{attribute 'GeneratedUsingTerminal: EK1122-0000-0018'}
{attribute addProperty BoxType "EK1122-0000-0018"}
{attribute addProperty Id "Beckhoff_EP7xxxsub_EK1100EK1100_1FC0878B2A_0001_EP7041_0002_0016EP7041_7A2D1F1A44A_0002_EP7041_0002_0017EP7041_7A2D1F1A44A_0003_EP7041_0002_0018EP7041_5C004D4E45A_0004_EP7041_0002_0019EP7041_5C004D4E45A_0005_EP7041_0002_0020EP7041_5C004D4E45A_0006_EP7041_0002_0021EP7041_5C004D4E45A_0007_EP7041_0002_0022EP7041_5C004D4E45A_0008_EP7041_0002_0023EP7041_5C004D4E45A_0009_EP7041_0002_0024EP7041_5C004D4E45A_0010_EP7041_0002_0025EP7041_5C004D4E45A_0011_EP7041_1002_0017EP7041_7A2D1F1A44A_0012_EP7041_1002_0018EP7041_5C004D4E45A_0013_EP7041_1002_0019EP7041_5C004D4E45A_0014_EP7041_1002_0020EP7041_5C004D4E45A_0015_EP7041_1002_0021EP7041_5C004D4E45A_0016_EP7041_1002_0022EP7041_5C004D4E45A_0017_EP7041_1002_0023EP7041_5C004D4E45A_0018_EP7041_1002_0024EP7041_5C004D4E45A_0019_EP7041_1002_0025EP7041_5C004D4E45A_0020_EP7041_2002_0016EP7041_5C004D4E45A_0021_EP7041_2002_0019EP7041_5C004D4E45A_0022_EP7041_2002_0020EP7041_5C004D4E45A_0023_EP7041_2002_0021EP7041_5C004D4E45A_0024_EP7041_2002_0022EP7041_5C004D4E45A_0025_EP7041_2002_0023EP7041_5C004D4E45A_0026_EP7041_2002_0024EP7041_5C004D4E45A_0027_EP7041_2002_0025EP7041_5C004D4E45A_0028_EP7041_3002_0016EP7041_B6E6359B46A_0029_EP7041_3002_0017EP7041_B6E6359B46A_0030_EP7041_3002_0018EP7041_B6E6359B46A_0031_EP7041_3002_0019EP7041_B6E6359B46A_0032_EP7041_3002_0020EP7041_B6E6359B46A_0033_EP7041_3002_0021EP7041_B6E6359B46A_0034_EP7041_3002_0022EP7041_B6E6359B46A_0035_EP7041_3102_0016EP7041_B6E6359B46A_0036_EP7041_3102_0017EP7041_B6E6359B46A_0037_EP7041_3102_0022EP7041_B6E6359B46A_0038_EP7047_1032_0021EP7047_B6E6359B46A_0039_EP7211_0034_0029EP7211_91DE43F025A_0040_EP7211_0034_0030EP7211_0985306B26A_0041_EP7211_0034_0031EP7211_0985306B26A_0042_EP7211_0034_0032EP7211_0985306B26A_0043_EP7211_0035_0029EP7211_24495B2825A_0044_EP7211_0035_0030EP7211_24495B2825A_0045_EP7211_0035_0031EP7211_24495B2825A_0046_EP7211_0035_0032EP7211_24495B2825A_0047_EP7342_0002_0016EP7342_A970B60778A_0048_EP7342_0002_0017EP7342_A970B60778A_0049_EP7342_0002_0018EP7342_A970B60778A_0050_EP7342_0002_0019EP7342_A970B60778A_0051_EP7342_0002_0020EP7342_A970B60778A_0052_EP7342_0002_0021EP7342_A970B60778A_0053_EP7342_0002_0022EP7342_A970B60778A_0054_EP7402_0057_0017A_0054_EP7402_0057_0017_470DA1C691"}
{attribute addProperty CRC "1867209835"}
{attribute addProperty Size "2560"}
TYPE Beckhoff_EP7xxxEK1122_6F4B5C6B EXTENDS EK1122_1FC0878B :
STRUCT
	{attribute addProperty Name "Beckhoff_EP7xxxsub_EK1100"}
	{attribute addProperty PreviousPort "Beckhoff EP7xxxEK1122 : D"}
	Beckhoff_EP7xxxsub_EK1100 : EK1100_1FC0878B;
	{attribute addProperty Name "A_0001_EP7041_0002_0016"}
	{attribute addProperty PreviousPort "Beckhoff EP7xxxsub EK1100 : C"}
	A_0001_EP7041_0002_0016 : EP7041_7A2D1F1A;
	{attribute addProperty Name "A_0002_EP7041_0002_0017"}
	{attribute addProperty PreviousPort "A_0001(EP7041-0002-0016) : B"}
	A_0002_EP7041_0002_0017 : EP7041_7A2D1F1A;
	{attribute addProperty Name "A_0003_EP7041_0002_0018"}
	{attribute addProperty PreviousPort "A_0002(EP7041-0002-0017) : B"}
	A_0003_EP7041_0002_0018 : EP7041_5C004D4E;
	{attribute addProperty Name "A_0004_EP7041_0002_0019"}
	{attribute addProperty PreviousPort "A_0003(EP7041-0002-0018) : B"}
	A_0004_EP7041_0002_0019 : EP7041_5C004D4E;
	{attribute addProperty Name "A_0005_EP7041_0002_0020"}
	{attribute addProperty PreviousPort "A_0004(EP7041-0002-0019) : B"}
	A_0005_EP7041_0002_0020 : EP7041_5C004D4E;
	{attribute addProperty Name "A_0006_EP7041_0002_0021"}
	{attribute addProperty PreviousPort "A_0005(EP7041-0002-0020) : B"}
	A_0006_EP7041_0002_0021 : EP7041_5C004D4E;
	{attribute addProperty Name "A_0007_EP7041_0002_0022"}
	{attribute addProperty PreviousPort "A_0006(EP7041-0002-0021) : B"}
	A_0007_EP7041_0002_0022 : EP7041_5C004D4E;
	{attribute addProperty Name "A_0008_EP7041_0002_0023"}
	{attribute addProperty PreviousPort "A_0007(EP7041-0002-0022) : B"}
	A_0008_EP7041_0002_0023 : EP7041_5C004D4E;
	{attribute addProperty Name "A_0009_EP7041_0002_0024"}
	{attribute addProperty PreviousPort "A_0008(EP7041-0002-0023) : B"}
	A_0009_EP7041_0002_0024 : EP7041_5C004D4E;
	{attribute addProperty Name "A_0010_EP7041_0002_0025"}
	{attribute addProperty PreviousPort "A_0009(EP7041-0002-0024) : B"}
	A_0010_EP7041_0002_0025 : EP7041_5C004D4E;
	{attribute addProperty Name "A_0011_EP7041_1002_0017"}
	{attribute addProperty PreviousPort "A_0010(EP7041-0002-0025) : B"}
	A_0011_EP7041_1002_0017 : EP7041_7A2D1F1A;
	{attribute addProperty Name "A_0012_EP7041_1002_0018"}
	{attribute addProperty PreviousPort "A_0011(EP7041-1002-0017) : B"}
	A_0012_EP7041_1002_0018 : EP7041_5C004D4E;
	{attribute addProperty Name "A_0013_EP7041_1002_0019"}
	{attribute addProperty PreviousPort "A_0012(EP7041-1002-0018) : B"}
	A_0013_EP7041_1002_0019 : EP7041_5C004D4E;
	{attribute addProperty Name "A_0014_EP7041_1002_0020"}
	{attribute addProperty PreviousPort "A_0013(EP7041-1002-0019) : B"}
	A_0014_EP7041_1002_0020 : EP7041_5C004D4E;
	{attribute addProperty Name "A_0015_EP7041_1002_0021"}
	{attribute addProperty PreviousPort "A_0014(EP7041-1002-0020) : B"}
	A_0015_EP7041_1002_0021 : EP7041_5C004D4E;
	{attribute addProperty Name "A_0016_EP7041_1002_0022"}
	{attribute addProperty PreviousPort "A_0015(EP7041-1002-0021) : B"}
	A_0016_EP7041_1002_0022 : EP7041_5C004D4E;
	{attribute addProperty Name "A_0017_EP7041_1002_0023"}
	{attribute addProperty PreviousPort "A_0016(EP7041-1002-0022) : B"}
	A_0017_EP7041_1002_0023 : EP7041_5C004D4E;
	{attribute addProperty Name "A_0018_EP7041_1002_0024"}
	{attribute addProperty PreviousPort "A_0017(EP7041-1002-0023) : B"}
	A_0018_EP7041_1002_0024 : EP7041_5C004D4E;
	{attribute addProperty Name "A_0019_EP7041_1002_0025"}
	{attribute addProperty PreviousPort "A_0018(EP7041-1002-0024) : B"}
	A_0019_EP7041_1002_0025 : EP7041_5C004D4E;
	{attribute addProperty Name "A_0020_EP7041_2002_0016"}
	{attribute addProperty PreviousPort "A_0019(EP7041-1002-0025) : B"}
	A_0020_EP7041_2002_0016 : EP7041_5C004D4E;
	{attribute addProperty Name "A_0021_EP7041_2002_0019"}
	{attribute addProperty PreviousPort "A_0020(EP7041-2002-0016) : B"}
	A_0021_EP7041_2002_0019 : EP7041_5C004D4E;
	{attribute addProperty Name "A_0022_EP7041_2002_0020"}
	{attribute addProperty PreviousPort "A_0021(EP7041-2002-0019) : B"}
	A_0022_EP7041_2002_0020 : EP7041_5C004D4E;
	{attribute addProperty Name "A_0023_EP7041_2002_0021"}
	{attribute addProperty PreviousPort "A_0022(EP7041-2002-0020) : B"}
	A_0023_EP7041_2002_0021 : EP7041_5C004D4E;
	{attribute addProperty Name "A_0024_EP7041_2002_0022"}
	{attribute addProperty PreviousPort "A_0023(EP7041-2002-0021) : B"}
	A_0024_EP7041_2002_0022 : EP7041_5C004D4E;
	{attribute addProperty Name "A_0025_EP7041_2002_0023"}
	{attribute addProperty PreviousPort "A_0024(EP7041-2002-0022) : B"}
	A_0025_EP7041_2002_0023 : EP7041_5C004D4E;
	{attribute addProperty Name "A_0026_EP7041_2002_0024"}
	{attribute addProperty PreviousPort "A_0025(EP7041-2002-0023) : B"}
	A_0026_EP7041_2002_0024 : EP7041_5C004D4E;
	{attribute addProperty Name "A_0027_EP7041_2002_0025"}
	{attribute addProperty PreviousPort "A_0026(EP7041-2002-0024) : B"}
	A_0027_EP7041_2002_0025 : EP7041_5C004D4E;
	{attribute addProperty Name "A_0028_EP7041_3002_0016"}
	{attribute addProperty PreviousPort "A_0027(EP7041-2002-0025) : B"}
	A_0028_EP7041_3002_0016 : EP7041_B6E6359B;
	{attribute addProperty Name "A_0029_EP7041_3002_0017"}
	{attribute addProperty PreviousPort "A_0028(EP7041-3002-0016) : B"}
	A_0029_EP7041_3002_0017 : EP7041_B6E6359B;
	{attribute addProperty Name "A_0030_EP7041_3002_0018"}
	{attribute addProperty PreviousPort "A_0029(EP7041-3002-0017) : B"}
	A_0030_EP7041_3002_0018 : EP7041_B6E6359B;
	{attribute addProperty Name "A_0031_EP7041_3002_0019"}
	{attribute addProperty PreviousPort "A_0030(EP7041-3002-0018) : B"}
	A_0031_EP7041_3002_0019 : EP7041_B6E6359B;
	{attribute addProperty Name "A_0032_EP7041_3002_0020"}
	{attribute addProperty PreviousPort "A_0031(EP7041-3002-0019) : B"}
	A_0032_EP7041_3002_0020 : EP7041_B6E6359B;
	{attribute addProperty Name "A_0033_EP7041_3002_0021"}
	{attribute addProperty PreviousPort "A_0032(EP7041-3002-0020) : B"}
	A_0033_EP7041_3002_0021 : EP7041_B6E6359B;
	{attribute addProperty Name "A_0034_EP7041_3002_0022"}
	{attribute addProperty PreviousPort "A_0033(EP7041-3002-0021) : B"}
	A_0034_EP7041_3002_0022 : EP7041_B6E6359B;
	{attribute addProperty Name "A_0035_EP7041_3102_0016"}
	{attribute addProperty PreviousPort "A_0034(EP7041-3002-0022) : B"}
	A_0035_EP7041_3102_0016 : EP7041_B6E6359B;
	{attribute addProperty Name "A_0036_EP7041_3102_0017"}
	{attribute addProperty PreviousPort "A_0035(EP7041-3102-0016) : B"}
	A_0036_EP7041_3102_0017 : EP7041_B6E6359B;
	{attribute addProperty Name "A_0037_EP7041_3102_0022"}
	{attribute addProperty PreviousPort "A_0036(EP7041-3102-0017) : B"}
	A_0037_EP7041_3102_0022 : EP7041_B6E6359B;
	{attribute addProperty Name "A_0038_EP7047_1032_0021"}
	{attribute addProperty PreviousPort "A_0037(EP7041-3102-0022) : B"}
	A_0038_EP7047_1032_0021 : EP7047_B6E6359B;
	{attribute addProperty Name "A_0039_EP7211_0034_0029"}
	{attribute addProperty PreviousPort "A_0038(EP7047-1032-0021) : B"}
	A_0039_EP7211_0034_0029 : EP7211_91DE43F0;
	{attribute addProperty Name "A_0040_EP7211_0034_0030"}
	{attribute addProperty PreviousPort "A_0039(EP7211-0034-0029) : B"}
	A_0040_EP7211_0034_0030 : EP7211_0985306B;
	{attribute addProperty Name "A_0041_EP7211_0034_0031"}
	{attribute addProperty PreviousPort "A_0040(EP7211-0034-0030) : B"}
	A_0041_EP7211_0034_0031 : EP7211_0985306B;
	{attribute addProperty Name "A_0042_EP7211_0034_0032"}
	{attribute addProperty PreviousPort "A_0041(EP7211-0034-0031) : B"}
	A_0042_EP7211_0034_0032 : EP7211_0985306B;
	{attribute addProperty Name "A_0043_EP7211_0035_0029"}
	{attribute addProperty PreviousPort "A_0042(EP7211-0034-0032) : B"}
	A_0043_EP7211_0035_0029 : EP7211_24495B28;
	{attribute addProperty Name "A_0044_EP7211_0035_0030"}
	{attribute addProperty PreviousPort "A_0043(EP7211-0035-0029) : B"}
	A_0044_EP7211_0035_0030 : EP7211_24495B28;
	{attribute addProperty Name "A_0045_EP7211_0035_0031"}
	{attribute addProperty PreviousPort "A_0044(EP7211-0035-0030) : B"}
	A_0045_EP7211_0035_0031 : EP7211_24495B28;
	{attribute addProperty Name "A_0046_EP7211_0035_0032"}
	{attribute addProperty PreviousPort "A_0045(EP7211-0035-0031) : B"}
	A_0046_EP7211_0035_0032 : EP7211_24495B28;
	{attribute addProperty Name "A_0047_EP7342_0002_0016"}
	{attribute addProperty PreviousPort "A_0046(EP7211-0035-0032) : B"}
	A_0047_EP7342_0002_0016 : EP7342_A970B607;
	{attribute addProperty Name "A_0048_EP7342_0002_0017"}
	{attribute addProperty PreviousPort "A_0047(EP7342-0002-0016) : B"}
	A_0048_EP7342_0002_0017 : EP7342_A970B607;
	{attribute addProperty Name "A_0049_EP7342_0002_0018"}
	{attribute addProperty PreviousPort "A_0048(EP7342-0002-0017) : B"}
	A_0049_EP7342_0002_0018 : EP7342_A970B607;
	{attribute addProperty Name "A_0050_EP7342_0002_0019"}
	{attribute addProperty PreviousPort "A_0049(EP7342-0002-0018) : B"}
	A_0050_EP7342_0002_0019 : EP7342_A970B607;
	{attribute addProperty Name "A_0051_EP7342_0002_0020"}
	{attribute addProperty PreviousPort "A_0050(EP7342-0002-0019) : B"}
	A_0051_EP7342_0002_0020 : EP7342_A970B607;
	{attribute addProperty Name "A_0052_EP7342_0002_0021"}
	{attribute addProperty PreviousPort "A_0051(EP7342-0002-0020) : B"}
	A_0052_EP7342_0002_0021 : EP7342_A970B607;
	{attribute addProperty Name "A_0053_EP7342_0002_0022"}
	{attribute addProperty PreviousPort "A_0052(EP7342-0002-0021) : B"}
	A_0053_EP7342_0002_0022 : EP7342_A970B607;
	{attribute addProperty Name "A_0054_EP7402_0057_0017"}
	{attribute addProperty PreviousPort "A_0053(EP7342-0002-0022) : B"}
	A_0054_EP7402_0057_0017 : A_0054_EP7402_0057_0017_470DA1C6;
END_STRUCT
END_TYPE

(* stored: Version 1.2.0.0, ProductVersion 3.1.4024.9
   DUT Beckhoff_EP7xxxEK1122_6F4B5C6B: Id {5c7ab07c-37bf-4804-9c77-d6fd33a5d2b4} *)
